FUNCTION_BLOCK DIV (* Divide *)
  (* Standard: 61499-2 *)
  (* Version 1.0, 02.01.2011, gsha041, UoA, Initial Version *)
  (* Compiler header: package fb.rt.UoA; *)
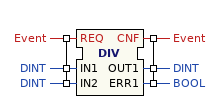
  EVENT_INPUT
    REQ WITH IN1, IN2; (* Normal Execution Request *)
  END_EVENT
  EVENT_OUTPUT
    CNF WITH OUT1, ERR1; (* Execution Confirmation *)
  END_EVENT
  VAR_INPUT
    IN1 : DINT; (* Dividend *)
    IN2 : DINT; (* Divisor *)
  END_VAR
  VAR_OUTPUT
    OUT1 : DINT; (* Result: INn1 / INn2 *)
    ERR1 : BOOL; (* Error (division by zero) *)
  END_VAR
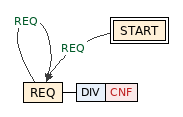
  EC_STATES
    START; (* Initial State *)
    REQ : DIV -> CNF; (* Normal execution *)
  END_STATES
  EC_TRANSITIONS
    START TO REQ := REQ;
    REQ TO REQ := REQ;
  END_TRANSITIONS
  ALGORITHM DIV IN ST: (* Normally executed algorithm *)
IF IN2 = 0 THEN
 ERR1 := true;
 ELSE
 OUT1 := IN1 / IN2;
 END_IF;
  END_ALGORITHM
END_FUNCTION_BLOCK
